FUNCTION "JsonW_LNK_Hello" : Void
{ S7_Optimized_Access := 'TRUE' }
VERSION : 0.1
   VAR_IN_OUT
      Buf : Array[*] of Byte;   // 출력 버퍼
      Pos : DInt;   // 다음 쓸 절대 인덱스 (< 0 = 오류 유지)
      Val : "LNK_Hello";   // 쓸 값
   END_VAR


BEGIN
	// GENERATED by gr-contract gen-link from "LNK_Hello" sig 16#BFAD9982 - do not edit
	// wire-spec 2 : 선언 순서, 공백 없음. 버퍼가 모자라면 Pos := LNK_JERR_OVERFLOW (끈끈한 오류, 호출자가 끝에 한 번 확인)
	"Json_WRaw"(Buf := #Buf, Pos := #Pos, Lit := '{"Plc":');
	"Json_WStr"(Buf := #Buf, Pos := #Pos, Val := #Val.Plc);
	"Json_WRaw"(Buf := #Buf, Pos := #Pos, Lit := ',"Proto":');
	"Json_WUSInt"(Buf := #Buf, Pos := #Pos, Val := #Val.Proto);
	"Json_WRaw"(Buf := #Buf, Pos := #Pos, Lit := ',"Formats":');
	"Json_WByte"(Buf := #Buf, Pos := #Pos, Val := #Val.Formats);
	"Json_WRaw"(Buf := #Buf, Pos := #Pos, Lit := ',"RegistryHash":');
	"Json_WDWord"(Buf := #Buf, Pos := #Pos, Val := #Val.RegistryHash);
	"Json_WRaw"(Buf := #Buf, Pos := #Pos, Lit := ',"HeartbeatMs":');
	"Json_WUDInt"(Buf := #Buf, Pos := #Pos, Val := #Val.HeartbeatMs);
	"Json_WRaw"(Buf := #Buf, Pos := #Pos, Lit := '}');
END_FUNCTION
